(* PLC project MQTT, OpenPLC MQTT 1.0, author OpenPLC Lib Writter *)
(* stored: creationDateTime 2023-04-26T04:54:00, modificationDateTime 2023-04-26T04:54:00 *)

(* Connects to the modbus tcp server with specified ADDRESS and PORT when CONNECT is set to TRUE. ADDRESS is STRING which can be represented as ipv4 (ex: 127.0.0.1) or as domain name (ex: www.google.com), default PORT is 502. REQ_TIMEOUT defines max waiting time to response after request. To change connection parameter you need to call MODBUS_TCP_DISCONNECT first. Upon a successful connection, SUCCESS is set to TRUE. *)
FUNCTION_BLOCK MODBUS_TCP_CONNECT
  VAR_INPUT
    CONNECT : BOOL;
    ADDRESS : STRING;
    PORT : UINT := 502;
    REQ_TIMEOUT : UINT;
  END_VAR
  VAR_OUTPUT
    SUCCESS : BOOL;
  END_VAR

            SUCCESS := 0;
          
END_FUNCTION_BLOCK

(* Reads coils using modbus (START_ADDRESS - address of first register, COUNT - registers count). If TCP set to true when connection to modbus tcp server will be used, otherwise modbus rtu will be used. Upon a successful operation, SUCCESS is set to TRUE and RESPONSE will be filled with requested values (each RESPONSE element type is BOOL, max ARRAY size is 128, indexes start from 0). *)
FUNCTION_BLOCK MODBUS_READ_COILS
  VAR_INPUT
    READ : BOOL;
    SLAVE_ID : USINT;
    START_ADDRESS : UINT;
    COUNT : UINT;
    TCP : BOOL;
  END_VAR
  VAR_OUTPUT
    SUCCESS : BOOL;
    RESPONSE : ARRAY[0..127] OF BOOL;
  END_VAR

            SUCCESS := 0;
          
END_FUNCTION_BLOCK

(* Reads discrete inputs using modbus (START_ADDRESS - address of first register, COUNT - registers count). If TCP set to true when connection to modbus tcp server will be used, otherwise modbus rtu will be used. Upon a successful operation, SUCCESS is set to TRUE and RESPONSE will be filled with requested values (each RESPONSE element type is BOOL, max ARRAY size is 128, indexes start from 0). *)
FUNCTION_BLOCK MODBUS_READ_DISCRETE_INPUTS
  VAR_INPUT
    READ : BOOL;
    SLAVE_ID : USINT;
    START_ADDRESS : UINT;
    COUNT : UINT;
    TCP : BOOL;
  END_VAR
  VAR_OUTPUT
    SUCCESS : BOOL;
    RESPONSE : ARRAY[0..127] OF BOOL;
  END_VAR

            SUCCESS := 0;
          
END_FUNCTION_BLOCK

(* Reads holding registers using modbus (START_ADDRESS - address of first register, COUNT - registers count). If TCP set to true when connection to modbus tcp server will be used, otherwise modbus rtu will be used. Upon a successful operation, SUCCESS is set to TRUE and RESPONSE will be filled with requested values (each RESPONSE element type is WORD, max ARRAY size is 128, indexes start from 0). *)
FUNCTION_BLOCK MODBUS_READ_HOLDING_REGISTERS
  VAR_INPUT
    READ : BOOL;
    SLAVE_ID : USINT;
    START_ADDRESS : UINT;
    COUNT : UINT;
    TCP : BOOL;
  END_VAR
  VAR_OUTPUT
    SUCCESS : BOOL;
    RESPONSE : ARRAY[0..127] OF WORD;
  END_VAR

            SUCCESS := 0;
          
END_FUNCTION_BLOCK

(* Reads input registers using modbus (START_ADDRESS - address of first register, COUNT - registers count). If TCP set to true when connection to modbus tcp server will be used, otherwise modbus rtu will be used. Upon a successful operation, SUCCESS is set to TRUE and RESPONSE will be filled with requested values (each RESPONSE element type is WORD, max ARRAY size is 128, indexes start from 0). *)
FUNCTION_BLOCK MODBUS_READ_INPUT_REGISTERS
  VAR_INPUT
    READ : BOOL;
    SLAVE_ID : USINT;
    START_ADDRESS : UINT;
    COUNT : UINT;
    TCP : BOOL;
  END_VAR
  VAR_OUTPUT
    SUCCESS : BOOL;
    RESPONSE : ARRAY[0..127] OF WORD;
  END_VAR

            SUCCESS := 0;
          
END_FUNCTION_BLOCK

(* Writes a new value to the specified modbus coil. If TCP set to true when connection to modbus tcp server will be used, otherwise modbus rtu will be used. Upon a successful operation, SUCCESS is set to TRUE. *)
FUNCTION_BLOCK MODBUS_WRITE_SINGLE_COIL
  VAR_INPUT
    WRITE : BOOL;
    SLAVE_ID : USINT;
    ADDRESS : UINT;
    NEW_VALUE : BOOL;
    TCP : BOOL;
  END_VAR
  VAR_OUTPUT
    SUCCESS : BOOL;
  END_VAR

            SUCCESS := 0;
          
END_FUNCTION_BLOCK

(* Writes a new value to the specified modbus register. If TCP set to true when connection to modbus tcp server will be used, otherwise modbus rtu will be used. Upon a successful operation, SUCCESS is set to TRUE. *)
FUNCTION_BLOCK MODBUS_WRITE_SINGLE_REGISTER
  VAR_INPUT
    WRITE : BOOL;
    SLAVE_ID : USINT;
    ADDRESS : UINT;
    NEW_VALUE : WORD;
    TCP : BOOL;
  END_VAR
  VAR_OUTPUT
    SUCCESS : BOOL;
  END_VAR

            SUCCESS := 0;
          
END_FUNCTION_BLOCK

(* Disconnects from current modbus tcp server when DISCONNECT is set to TRUE. Upon a successful disconnection, SUCCESS is set to TRUE. *)
FUNCTION_BLOCK MODBUS_TCP_DISCONNECT
  VAR_INPUT
    DISCONNECT : BOOL;
  END_VAR
  VAR_OUTPUT
    SUCCESS : BOOL;
  END_VAR

  SUCCESS := 0;
END_FUNCTION_BLOCK
